// TIA Portal V19 export
TYPE "IFM_PN3594_IO"
TITLE = PN3594 DeviceID: 431 Vendor:310
   STRUCT
      Addr : Int;   // IO Address
      Value : Real;   // Pressure_Bar
      DeviceStatus : Byte;   // Device Status
      OUT1 : Bool;   // Out 1
      OUT2 : Bool;   // Out 2
      O_DI4 : Bool;   // Port pin 4
      O_DI2 : Bool;   // Port pin 2
      O_DA : Bool;   // Device Attached
      O_DE : Bool;   // Device Error
      O_PQ : Bool;   // Value Valid
   END_STRUCT;
END_TYPE
